Universal Robots PolyScope program: proyecto_jz.urp

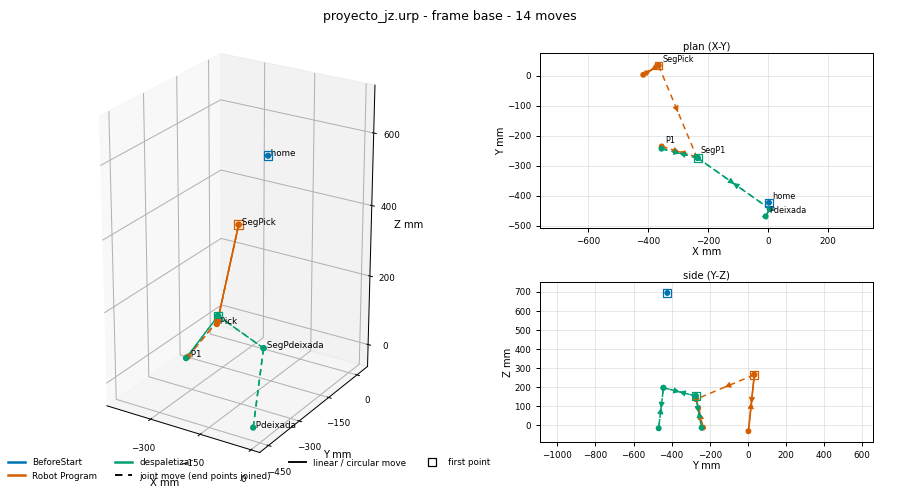
[picture p0: tool path of proyecto_jz.urp in frame base, 14 of 14 moves have a stored position in this frame; points joined in program order, loops and branches not executed]
Program proyecto_jz (installation=default directory=/programs createdIn=5.9.3.1031212 lastSavedIn=5.9.3.1031212 robotSerialNumber=20195300809)
Calibrated DH parameters: a=[-0.000085, -0.20076, -0.212369, 0.000121, -0.000118, 0]; d=[0.15185, -26.306375, 24.753047, 1.684739, 0.085386, 0.092088]; alpha=[1.572149, -0.00522, -0.011864, 1.571339, -1.571085, 0]; deltaTheta=[0, 0.599885, -0.513355, -0.086555, 0.000006, 0]
BeforeStart
  MoveJ speed 60 deg/s, acceleration 80 deg/s^2 (useActiveTCP=true) feature=Base
    Waypoint home: TCP in base x=2.912 y=-422.717 z=694.835 mm, rx=-0.0077 ry=2.2126 rz=-2.219 rad; joints [-0.428, -89.93, 0.173, -90.508, 0.025, 0.392] deg; TCP offset x=0 y=0 z=200 mm, rx=0 ry=0 rz=0 rad
  URCap Gripper Activate (Robotiq_Grippers, Robotiq Inc.) dataModel(ResetAndActivateKey=false)
  URCap Gripper (Robotiq_Grippers, Robotiq Inc.) dataModel(position=0.0, force=0.0, speed=0.0, positionInDouble=0.0, forceInDouble=0.0, speedInDouble=0.0, slaveIds=[9], blocking=true)
  cont := 1
Robot Program (runOnlyOnce=false)
  Folder recollida
    MoveJ speed 60 deg/s, acceleration 80 deg/s^2 (useActiveTCP=true) feature=Base
      Waypoint SegPick: TCP in base x=-364.863 y=34.133 z=265.269 mm, rx=-2.148 ry=-1.8737 rz=0.2024 rad; joints [-27.989, -92.053, 57.843, -73.916, -89.13, -19.601] deg
    MoveL speed 250 mm/s, acceleration 1200 mm/s^2 (useActiveTCP=true) feature=Base
      Waypoint Pick: TCP in base x=-415.778 y=3.266 z=-31.153 mm, rx=-2.2658 ry=-2.1292 rz=-0.0005 rad; joints [-18.243, -61.038, 91.452, -122.057, -91.64, -15.01] deg
      URCap Gripper (Robotiq_Grippers, Robotiq Inc.) dataModel(position=100.0, force=0.0, speed=0.0, positionInDouble=100.0, forceInDouble=0.0, speedInDouble=0.0, slaveIds=[9], blocking=true)
      Waypoint SegPick: TCP in base x=-364.863 y=34.133 z=265.269 mm, rx=-2.148 ry=-1.8737 rz=0.2024 rad; joints [-27.989, -92.053, 57.843, -73.916, -89.13, -19.601] deg
    If cont≟9
      cont := 1
      Call despaletizar
    URCap Palletizing (pallet-impl, Universal Robots) dataModel(palletFeature=Base, isPalletizing=true, rememberTraversal=true, afterSelected=false, beforeSelected=false, Variable(key=name, variable(name=Pallet_1)), Variable(key=layerNumberVariable, variable(name=Pallet_1_lno, initializeExpression=1)), Variable(key=layerCountingVariable, variable(name=Pallet_1_lct, initializeExpression=1)), Variable(key=handleSeparatorVariable, variable(name=Pallet_1_sep, initializeExpression=False)), Variable(key=totalCountVariable, variable(name=Pallet_1_tct, initializeExpression=1)), Variable(key=referencePoint, variable(featureName=referencePoint)), Variable(key=separatorPoint, variable(featureName=separatorPoint)), Length(key=objectHeight value=0.002 unit=M), Variable(key=globalCountingVariable, variable=Pallet_1_cnt)); state(isChildrenLocked=true)
      URCap Patterns (pallet-impl, Universal Robots) state(isChildrenLocked=true)
        URCap Pattern (pallet-impl, Universal Robots) dataModel(UUID=5f113852-ae8f-4cc2-91b8-8522b6a8a6a4, patternType=GRID, columns=3, rows=3, Variable(key=nameVariable, variable(name=Grid_Pattern_1))); state(isChildrenLocked=true)
          URCap Item (pallet-impl, Universal Robots) dataModel(UUID=20d84a79-391a-4d00-bace-49f084b26c2f, patternType=GRID, index=0, calibrationDeltaTheta=[2.0871938292282843E-8, 0.5998849625986696, -0.513354759222901, -0.08655474087847535, 6.239817607139875E-6, -6.658617090343766E-8], calibrationA=[-8.52060452638757E-5, -0.2007601879611388, -0.2123691625519033, 1.2105607098011576E-4, -1.1833705743435544E-4, 0.0], calibrationD=[0.15184970286177432, -26.306374840159272, 24.75304670983349, 1.6847390881089916, 0.085385969004481, 0.09208826337351553], calibrationAlpha=[1.5721487795181908, -0.005219907129425837, -0.011864150755780208, 1.5713392161993658, -1.5710853432049288, 0.0], calibrationJointChecksum=[-1860213401, -1859864814, -1494669377, -1328152407, -1329437658, -1329056899], calibrationStatus=2, calibrationValidChecksum=true, baseToFeature=[0.0, 0.0, 0.0, 0.0, 0.0, 0.0], TCPOffset=[1.4143476017108858E-5, 2.345864315134172E-6, 0.2000068177482045, -3.170362765922186E-5, 2.0357059619337508E-5, 4.753924383008288E-5], Variable(key=variable, variable(name=CornerItem_1)), JointPositions(key=jointpositions, JointPosition(key=[1], Angle(key=pos value=0.273712 unit=RAD)), JointPosition(key=[2], Angle(key=pos value=-1.027217 unit=RAD)), JointPosition(key=[3], Angle(key=pos value=1.4787 unit=RAD)), JointPosition(key=[4], Angle(key=pos value=-2.013475 unit=RAD)), JointPosition(key=[5], Angle(key=pos value=-1.585729 unit=RAD)), JointPosition(key=[6], Angle(key=pos value=0.253209 unit=RAD))))
          URCap Item (pallet-impl, Universal Robots) dataModel(UUID=1dfddf64-9e06-4662-ad2b-a4af7187a8de, patternType=GRID, index=1, calibrationDeltaTheta=[2.0871938292282843E-8, 0.5998849625986696, -0.513354759222901, -0.08655474087847535, 6.239817607139875E-6, -6.658617090343766E-8], calibrationA=[-8.52060452638757E-5, -0.2007601879611388, -0.2123691625519033, 1.2105607098011576E-4, -1.1833705743435544E-4, 0.0], calibrationD=[0.15184970286177432, -26.306374840159272, 24.75304670983349, 1.6847390881089916, 0.085385969004481, 0.09208826337351553], calibrationAlpha=[1.5721487795181908, -0.005219907129425837, -0.011864150755780208, 1.5713392161993658, -1.5710853432049288, 0.0], calibrationJointChecksum=[-1860213401, -1859864814, -1494669377, -1328152407, -1329437658, -1329056899], calibrationStatus=2, calibrationValidChecksum=true, baseToFeature=[0.0, 0.0, 0.0, 0.0, 0.0, 0.0], TCPOffset=[-9.336587432795529E-6, 1.13081380309632E-5, 0.2000075440100896, -3.1098400745511366E-5, -1.1867751621430461E-5, -1.3229802096909477E-5], Variable(key=variable, variable(name=CornerItem_2)), JointPositions(key=jointpositions, JointPosition(key=[1], Angle(key=pos value=0.516711 unit=RAD)), JointPosition(key=[2], Angle(key=pos value=-1.595201 unit=RAD)), JointPosition(key=[3], Angle(key=pos value=2.28614 unit=RAD)), JointPosition(key=[4], Angle(key=pos value=-2.286332 unit=RAD)), JointPosition(key=[5], Angle(key=pos value=-1.623689 unit=RAD)), JointPosition(key=[6], Angle(key=pos value=0.452308 unit=RAD))))
          URCap Item (pallet-impl, Universal Robots) dataModel(UUID=edffe996-6e7e-4cd1-8c05-ba43609d1eb9, patternType=GRID, index=2, calibrationDeltaTheta=[2.0871938292282843E-8, 0.5998849625986696, -0.513354759222901, -0.08655474087847535, 6.239817607139875E-6, -6.658617090343766E-8], calibrationA=[-8.52060452638757E-5, -0.2007601879611388, -0.2123691625519033, 1.2105607098011576E-4, -1.1833705743435544E-4, 0.0], calibrationD=[0.15184970286177432, -26.306374840159272, 24.75304670983349, 1.6847390881089916, 0.085385969004481, 0.09208826337351553], calibrationAlpha=[1.5721487795181908, -0.005219907129425837, -0.011864150755780208, 1.5713392161993658, -1.5710853432049288, 0.0], calibrationJointChecksum=[-1860213401, -1859864814, -1494669377, -1328152407, -1329437658, -1329056899], calibrationStatus=2, calibrationValidChecksum=true, baseToFeature=[0.0, 0.0, 0.0, 0.0, 0.0, 0.0], TCPOffset=[-8.863471887721186E-6, 2.6791358828714973E-5, 0.2000185994487076, -6.311902562673469E-5, 1.2356726224438938E-5, -8.825275738171846E-6], Variable(key=variable, variable(name=CornerItem_3)), JointPositions(key=jointpositions, JointPosition(key=[1], Angle(key=pos value=0.464245 unit=RAD)), JointPosition(key=[2], Angle(key=pos value=-0.8816 unit=RAD)), JointPosition(key=[3], Angle(key=pos value=1.275658 unit=RAD)), JointPosition(key=[4], Angle(key=pos value=-2.07629 unit=RAD)), JointPosition(key=[5], Angle(key=pos value=-1.529262 unit=RAD)), JointPosition(key=[6], Angle(key=pos value=0.432238 unit=RAD))))
          URCap Item (pallet-impl, Universal Robots) dataModel(UUID=7ed241a1-7805-46f5-b879-d77fd2d795ad, patternType=GRID, index=3, calibrationDeltaTheta=[2.0871938292282843E-8, 0.5998849625986696, -0.513354759222901, -0.08655474087847535, 6.239817607139875E-6, -6.658617090343766E-8], calibrationA=[-8.52060452638757E-5, -0.2007601879611388, -0.2123691625519033, 1.2105607098011576E-4, -1.1833705743435544E-4, 0.0], calibrationD=[0.15184970286177432, -26.306374840159272, 24.75304670983349, 1.6847390881089916, 0.085385969004481, 0.09208826337351553], calibrationAlpha=[1.5721487795181908, -0.005219907129425837, -0.011864150755780208, 1.5713392161993658, -1.5710853432049288, 0.0], calibrationJointChecksum=[-1860213401, -1859864814, -1494669377, -1328152407, -1329437658, -1329056899], calibrationStatus=2, calibrationValidChecksum=true, baseToFeature=[0.0, 0.0, 0.0, 0.0, 0.0, 0.0], TCPOffset=[-1.6657031478739537E-5, 8.483564769096175E-6, 0.199999786663717, -3.539693042070147E-5, -5.019841375289947E-5, 2.787065139229695E-7], Variable(key=variable, variable(name=CornerItem_4)), JointPositions(key=jointpositions, JointPosition(key=[1], Angle(key=pos value=0.784683 unit=RAD)), JointPosition(key=[2], Angle(key=pos value=-1.186045 unit=RAD)), JointPosition(key=[3], Angle(key=pos value=1.695681 unit=RAD)), JointPosition(key=[4], Angle(key=pos value=-2.019179 unit=RAD)), JointPosition(key=[5], Angle(key=pos value=-1.595366 unit=RAD)), JointPosition(key=[6], Angle(key=pos value=0.820315 unit=RAD))))
      URCap Layers (pallet-impl, Universal Robots) dataModel(separators=[false], selectedPatterns=[5f113852-ae8f-4cc2-91b8-8522b6a8a6a4])
      URCap At Each Item (pallet-impl, Universal Robots) dataModel(currentWizardState=MANUAL)
        MoveJ speed 60 deg/s, acceleration 80 deg/s^2 (useActiveTCP=true) feature=Base
          Waypoint SegP1: TCP in base x=-237.599 y=-270.684 z=137.402 mm, rx=2.0585 ry=2.287 rz=-0.2081 rad; joints [21.445, -90.968, 85.19, -89.722, -84.385, 15.89] deg
          Waypoint P1: TCP in base x=-354.373 y=-235.325 z=-12.164 mm, rx=2.1426 ry=2.2822 rz=-0.0416 rad; joints [14.578, -61.152, 85.597, -115.412, -89.438, 10.732] deg
          URCap Gripper (Robotiq_Grippers, Robotiq Inc.) dataModel(position=0.0, force=0.0, speed=0.0, positionInDouble=0.0, forceInDouble=0.0, speedInDouble=0.0, slaveIds=[9], blocking=true)
          Waypoint SegP1: TCP in base x=-237.599 y=-270.684 z=137.402 mm, rx=2.0585 ry=2.287 rz=-0.2081 rad; joints [21.445, -90.968, 85.19, -89.722, -84.385, 15.89] deg
SubProgram -> despaletizar
SubProgram despaletizar (keepSynchronizedWithDisk=false)
  URCap Palletizing (pallet-impl, Universal Robots) dataModel(palletFeature=Base, isPalletizing=false, rememberTraversal=true, Variable(key=name, variable(name=Pallet_2)), Variable(key=layerNumberVariable, variable(name=Pallet_2_lno, initializeExpression=1)), Variable(key=layerCountingVariable, variable(name=Pallet_2_lct, initializeExpression=1)), Variable(key=handleSeparatorVariable, variable(name=Pallet_2_sep, initializeExpression=False)), Variable(key=totalCountVariable, variable(name=Pallet_2_tct, initializeExpression=1)), Variable(key=referencePoint, variable(featureName=referencePoin_1)), Variable(key=separatorPoint, variable(featureName=separatorPoin_1)), Length(key=objectHeight value=0.002 unit=M), Variable(key=globalCountingVariable, variable=Pallet_2_cnt)); state(isChildrenLocked=true)
    URCap Patterns (pallet-impl, Universal Robots) state(isChildrenLocked=true)
      URCap Pattern (pallet-impl, Universal Robots) dataModel(UUID=2779d410-9d27-4111-a702-48ef58dcf734, patternType=GRID, columns=3, rows=3, Variable(key=nameVariable, variable(name=Grid_Pattern_2))); state(isChildrenLocked=true)
        URCap Item (pallet-impl, Universal Robots) dataModel(UUID=c37c83a6-6329-4650-9a46-550b1b4faa2f, patternType=GRID, index=0, calibrationDeltaTheta=[2.0871938292282843E-8, 0.5998849625986696, -0.513354759222901, -0.08655474087847535, 6.239817607139875E-6, -6.658617090343766E-8], calibrationA=[-8.52060452638757E-5, -0.2007601879611388, -0.2123691625519033, 1.2105607098011576E-4, -1.1833705743435544E-4, 0.0], calibrationD=[0.15184970286177432, -26.306374840159272, 24.75304670983349, 1.6847390881089916, 0.085385969004481, 0.09208826337351553], calibrationAlpha=[1.5721487795181908, -0.005219907129425837, -0.011864150755780208, 1.5713392161993658, -1.5710853432049288, 0.0], calibrationJointChecksum=[-1860213401, -1859864814, -1494669377, -1328152407, -1329437658, -1329056899], calibrationStatus=2, calibrationValidChecksum=true, baseToFeature=[0.0, 0.0, 0.0, 0.0, 0.0, 0.0], TCPOffset=[-7.614389200105709E-6, 2.235433198710668E-5, 0.20002024586167785, -6.116884634854972E-5, 2.6543668956451573E-6, -2.41083690342031E-7], Variable(key=variable, variable(name=CornerItem_5)), JointPositions(key=jointpositions, JointPosition(key=[1], Angle(key=pos value=0.271737 unit=RAD)), JointPosition(key=[2], Angle(key=pos value=-1.092419 unit=RAD)), JointPosition(key=[3], Angle(key=pos value=1.598679 unit=RAD)), JointPosition(key=[4], Angle(key=pos value=-2.12611 unit=RAD)), JointPosition(key=[5], Angle(key=pos value=-1.58755 unit=RAD)), JointPosition(key=[6], Angle(key=pos value=0.24438 unit=RAD))))
        URCap Item (pallet-impl, Universal Robots) dataModel(UUID=f987b466-d91e-454b-9ea9-98f03afa6eb1, patternType=GRID, index=1, calibrationDeltaTheta=[2.0871938292282843E-8, 0.5998849625986696, -0.513354759222901, -0.08655474087847535, 6.239817607139875E-6, -6.658617090343766E-8], calibrationA=[-8.52060452638757E-5, -0.2007601879611388, -0.2123691625519033, 1.2105607098011576E-4, -1.1833705743435544E-4, 0.0], calibrationD=[0.15184970286177432, -26.306374840159272, 24.75304670983349, 1.6847390881089916, 0.085385969004481, 0.09208826337351553], calibrationAlpha=[1.5721487795181908, -0.005219907129425837, -0.011864150755780208, 1.5713392161993658, -1.5710853432049288, 0.0], calibrationJointChecksum=[-1860213401, -1859864814, -1494669377, -1328152407, -1329437658, -1329056899], calibrationStatus=2, calibrationValidChecksum=true, baseToFeature=[0.0, 0.0, 0.0, 0.0, 0.0, 0.0], TCPOffset=[6.778131657919628E-6, 5.576424972453253E-6, 0.20000501384239094, -2.309727936605139E-5, 3.652058883038196E-5, -4.676423738777179E-7], Variable(key=variable, variable(name=CornerItem_6)), JointPositions(key=jointpositions, JointPosition(key=[1], Angle(key=pos value=0.479153 unit=RAD)), JointPosition(key=[2], Angle(key=pos value=-1.593027 unit=RAD)), JointPosition(key=[3], Angle(key=pos value=2.237964 unit=RAD)), JointPosition(key=[4], Angle(key=pos value=-2.230715 unit=RAD)), JointPosition(key=[5], Angle(key=pos value=-1.588713 unit=RAD)), JointPosition(key=[6], Angle(key=pos value=0.426885 unit=RAD))))
        URCap Item (pallet-impl, Universal Robots) dataModel(UUID=3823b940-1985-43ef-81c7-1d96114db9d2, patternType=GRID, index=2, calibrationDeltaTheta=[2.0871938292282843E-8, 0.5998849625986696, -0.513354759222901, -0.08655474087847535, 6.239817607139875E-6, -6.658617090343766E-8], calibrationA=[-8.52060452638757E-5, -0.2007601879611388, -0.2123691625519033, 1.2105607098011576E-4, -1.1833705743435544E-4, 0.0], calibrationD=[0.15184970286177432, -26.306374840159272, 24.75304670983349, 1.6847390881089916, 0.085385969004481, 0.09208826337351553], calibrationAlpha=[1.5721487795181908, -0.005219907129425837, -0.011864150755780208, 1.5713392161993658, -1.5710853432049288, 0.0], calibrationJointChecksum=[-1860213401, -1859864814, -1494669377, -1328152407, -1329437658, -1329056899], calibrationStatus=2, calibrationValidChecksum=true, baseToFeature=[0.0, 0.0, 0.0, 0.0, 0.0, 0.0], TCPOffset=[1.900423207573665E-5, 5.534967785769673E-6, 0.20003286617141142, -6.667816233336303E-5, 2.7807149137424984E-5, 4.9107784141547554E-5], Variable(key=variable, variable(name=CornerItem_7)), JointPositions(key=jointpositions, JointPosition(key=[1], Angle(key=pos value=0.497316 unit=RAD)), JointPosition(key=[2], Angle(key=pos value=-0.873648 unit=RAD)), JointPosition(key=[3], Angle(key=pos value=1.260064 unit=RAD)), JointPosition(key=[4], Angle(key=pos value=-2.051824 unit=RAD)), JointPosition(key=[5], Angle(key=pos value=-1.581222 unit=RAD)), JointPosition(key=[6], Angle(key=pos value=0.49869 unit=RAD))))
        URCap Item (pallet-impl, Universal Robots) dataModel(UUID=fd6f6c5a-33d5-4043-8905-a1821ed65b9f, patternType=GRID, index=3, calibrationDeltaTheta=[2.0871938292282843E-8, 0.5998849625986696, -0.513354759222901, -0.08655474087847535, 6.239817607139875E-6, -6.658617090343766E-8], calibrationA=[-8.52060452638757E-5, -0.2007601879611388, -0.2123691625519033, 1.2105607098011576E-4, -1.1833705743435544E-4, 0.0], calibrationD=[0.15184970286177432, -26.306374840159272, 24.75304670983349, 1.6847390881089916, 0.085385969004481, 0.09208826337351553], calibrationAlpha=[1.5721487795181908, -0.005219907129425837, -0.011864150755780208, 1.5713392161993658, -1.5710853432049288, 0.0], calibrationJointChecksum=[-1860213401, -1859864814, -1494669377, -1328152407, -1329437658, -1329056899], calibrationStatus=2, calibrationValidChecksum=true, baseToFeature=[0.0, 0.0, 0.0, 0.0, 0.0, 0.0], TCPOffset=[-1.1154836254689826E-7, -5.044126224290624E-6, 0.19999894331173282, 1.7183751531910354E-5, -4.6008594287543733E-7, -1.1521265761763123E-5], Variable(key=variable, variable(name=CornerItem_8)), JointPositions(key=jointpositions, JointPosition(key=[1], Angle(key=pos value=0.784335 unit=RAD)), JointPosition(key=[2], Angle(key=pos value=-1.210527 unit=RAD)), JointPosition(key=[3], Angle(key=pos value=1.760906 unit=RAD)), JointPosition(key=[4], Angle(key=pos value=-2.095719 unit=RAD)), JointPosition(key=[5], Angle(key=pos value=-1.602761 unit=RAD)), JointPosition(key=[6], Angle(key=pos value=0.792535 unit=RAD))))
    URCap Layers (pallet-impl, Universal Robots) dataModel(separators=[false], selectedPatterns=[2779d410-9d27-4111-a702-48ef58dcf734])
    URCap At Each Item (pallet-impl, Universal Robots) dataModel(currentWizardState=MANUAL)
      MoveJ speed 60 deg/s, acceleration 80 deg/s^2 (useActiveTCP=true) feature=Base
        Waypoint SegP2: TCP in base x=-234.505 y=-273.821 z=153.642 mm, rx=2.0242 ry=2.3218 rz=-0.1467 rad; joints [23.115, -87.17, 75.747, -82.09, -85.443, 15.68] deg
        Waypoint P2: TCP in base x=-355.056 y=-242.774 z=-13.22 mm, rx=-2.1613 ry=-2.2629 rz=-0.0075 rad; joints [17.07, -58.39, 81.028, -112.765, -91.551, 14.212] deg
        URCap Gripper (Robotiq_Grippers, Robotiq Inc.) dataModel(position=0.0, force=0.0, speed=0.0, positionInDouble=0.0, forceInDouble=0.0, speedInDouble=0.0, slaveIds=[9], blocking=true)
        URCap Gripper (Robotiq_Grippers, Robotiq Inc.) dataModel(position=100.0, force=0.0, speed=0.0, positionInDouble=100.0, forceInDouble=0.0, speedInDouble=0.0, slaveIds=[9], blocking=true)
        Waypoint SegP2: TCP in base x=-234.505 y=-273.821 z=153.642 mm, rx=2.0242 ry=2.3218 rz=-0.1467 rad; joints [23.115, -87.17, 75.747, -82.09, -85.443, 15.68] deg
        Waypoint SegPdeixada: TCP in base x=5.415 y=-443.256 z=196.939 mm, rx=-0.3111 ry=-3.0584 rz=0.5059 rad; joints [71.585, -80.769, 66.473, -94.3, -88.294, -6.356] deg
        Waypoint Pdeixada: TCP in base x=-8.355 y=-468.085 z=-15.948 mm, rx=-0.1881 ry=-3.1321 rz=0.0749 rad; joints [72.334, -52.196, 72.517, -113.029, -90.304, -11.048] deg
        URCap Gripper (Robotiq_Grippers, Robotiq Inc.) dataModel(position=0.0, force=0.0, speed=0.0, positionInDouble=0.0, forceInDouble=0.0, speedInDouble=0.0, slaveIds=[9], blocking=true)
        Waypoint SegPdeixada: TCP in base x=5.415 y=-443.256 z=196.939 mm, rx=-0.3111 ry=-3.0584 rz=0.5059 rad; joints [71.585, -80.769, 66.473, -94.3, -88.294, -6.356] deg
        Waypoint SegP2: TCP in base x=-234.505 y=-273.821 z=153.642 mm, rx=2.0242 ry=2.3218 rz=-0.1467 rad; joints [23.115, -87.17, 75.747, -82.09, -85.443, 15.68] deg
